FUNCTION alg_a_x: BOOL
VAR_INPUT
    state: STATE;
END_VAR

alg_a_x := TRUE;

END_FUNCTION

(* stored: ProductVersion 3.1.0.18, Version 1.1.0.1 *)
